FUNCTION_BLOCK Aborting_State  IMPLEMENTS ITF_State
VAR_INPUT
END_VAR
VAR_OUTPUT
END_VAR
VAR
	pPML_Base : POINTER TO PML_StatePattern_Base;
	_stateMachine : IPmlStateMachine;
END_VAR

METHOD Cycle : BOOL
_stateMachine.SetStateComplete();
pPML_Base^.SetState(pPML_Base^.aborted);
END_METHOD

METHOD FB_init : BOOL
VAR_INPUT
	bInitRetains : BOOL; // if TRUE, the retain variables are initialized (warm start / cold start)
	bInCopyCode : BOOL;  // if TRUE, the instance afterwards gets moved into the copy code (online change)
	pPML_Base : POINTER TO PML_StatePattern_Base;
	statemachine : IPmlStateMachine;
END_VAR
_stateMachine := statemachine;
THIS^.pPML_Base := pPML_Base;
END_METHOD

END_FUNCTION_BLOCK

(* stored: Version 1.1.0.1, ProductVersion 3.1.4024.11
   POU Aborting_State: Id {efef8688-79a1-4985-bd2c-9f23761f91b9}, SpecialFunc None
   Method Cycle: Id {ef9f4632-e6d8-4187-96e3-a3c4a4d5873f}
   Method FB_init: Id {a93f572d-56b6-4db2-858b-602a3a4a7f42} *)
